KUKA KRL program: nplacestr6RS1.src, nplacestr6RS1.dat

--- nplacestr6RS1.src ---
&ACCESS RVP
&REL 1
&PARAM TEMPLATE = C:\KRC\Roboter\Template\ExpertVorgabe
&PARAM EDITMASK = *
DEF nplacestr6RS1( )
;FOLD INI
  ;FOLD BASISTECH INI
    GLOBAL INTERRUPT DECL 3 WHEN $STOPMESS==TRUE DO IR_STOPM ( )
    INTERRUPT ON 3
    BAS (#INITMOV,0 )
  ;ENDFOLD (BASISTECH INI)
  ;FOLD USER INI
    ;Make your modifications here

  ;ENDFOLD (USER INI)
;ENDFOLD (INI)




SWITCH NumCuring

;*******************************************************
CASE 90613
;*******************************************************
;*** Utilizar para hacer touchup en ptp a continuacion ***;
; 1  Ejecutar Axis_Rob_Move
; 2  Hacer TouchUp en ptp
; 3  Eliminar Axis_Rob_Move y comentarios

Axis_Rob_Move(1.69,-82.8,66.93,14.32,12.14,193,70,50)

;FOLD PTP pWB90613RS1 Vel=100 % PDAT_MESA Tool[10]:AMF1_G1000 Base[14]:BWB2S1;%{PE}%R 5.5.32,%MKUKATPBASIS,%CMOVE,%VPTP,%P 1:PTP, 2:pWB90613RS1, 3:, 5:100, 7:PDAT_MESA
$BWDSTART=FALSE
PDAT_ACT=PPDAT_MESA
FDAT_ACT=FpWB90613RS1
BAS(#PTP_PARAMS,100)
PTP XpWB90613RS1
;ENDFOLD
;*********************************************************;

;***Axis_Rob_Move de ayuda para aproximarse a dejada ***;
; Borrar tras touchup en LIN de dejada
Axis_Rob_Move(-90.22,-57.13,49.23,-5.44,97.37,193.9,20,50)
;*******************************************************;

PTP_OFFS(XP90613RS1, FP90613RS1, 0, -450, 30, 0, 0, 0, #TOOL, 20, 50, 0.0)

Cicle_Grp_M1000 (Inic_Pla_Right)

;***borrar***;
cyltopos(prg_200)
halt
;************;

LIN_OFFS(XP90613RS1, FP90613RS1, 0, 0, 30, 0, 0, 0, #TOOL, 0.1, 50, 0.0)
LIN_OFFS(XP90613RS1, FP90613RS1, 0, 0, 15, 0, 0, 0, #TOOL, 0.1, 50, 0.0)

Cntr_Grp_M1000 (C05C06,RH)

;FOLD LIN P90613RS1 Vel=0.1 m/s LV020Z0 Tool[10]:AMF1_G1000 Base[14]:BWB2S1;%{PE}%R 5.5.32,%MKUKATPBASIS,%CMOVE,%VLIN,%P 1:LIN, 2:P90613RS1, 3:, 5:0.1, 7:V020Z0
$BWDSTART=FALSE
LDAT_ACT=LV020Z0
FDAT_ACT=FP90613RS1
BAS(#CP_PARAMS,0.1)
LIN XP90613RS1
;ENDFOLD

Cntr_Grp_M1000 (AMF09,RLS)
Cyltopos (PRG_51)
Cntr_Grp_M1000 (C07C08,RH)
Cyltopos (PRG_61)
Cntr_Grp_M1000 (AMF10,RLS)
Cntr_Grp_M1000 (C05C06,FREE)
Cntr_Grp_M1000 (C07C08,FREE)
Cyltopos(PRG_88)
LIN_REL{Z -20}#TOOL
Cyltopos (PRG_105)
LIN_REL{Z -30}#TOOL
Cyltopos (PRG_200)

;*** MOVIMIENTOS DE OFFSETS ***;

LIN_OFFS(XP90613RS1, FP90613RS1, 0, 0, -50, 0, 0, 0, #TOOL, 0.3, 50, 0.0)
LIN_OFFS(XP90613RS1, FP90613RS1, 0, -450, -50, 0, 0, 0, #TOOL, 0.3, 50, 0.0)


;******* MEDICION LASER *******;

LIN_OFFS(XPLAS90613RS1_1, FPLAS90613RS1_1, 0, -200, 0, 0, 0, 0, #TOOL, 0.3, 50, 0.0)

cyltopos (prg_61)

;FOLD LIN PLAS90613RS1_1 Vel=0.3 m/s LV020Z0 Tool[10]:AMF1_G1000 Base[14]:BWB2S1;%{PE}%R 5.5.32,%MKUKATPBASIS,%CMOVE,%VLIN,%P 1:LIN, 2:PLAS90613RS1_1, 3:, 5:0.3, 7:V020Z0
$BWDSTART=FALSE
LDAT_ACT=LV020Z0
FDAT_ACT=FPLAS90613RS1_1
BAS(#CP_PARAMS,0.3)
LIN XPLAS90613RS1_1
;ENDFOLD

;Movimimiento de busqueda con laser
;Search( , )

;FOLD LIN PLAS90613RS1_2 Vel=0.3 m/s LV020Z0 Tool[10]:AMF1_G1000 Base[14]:BWB2S1;%{PE}%R 5.5.32,%MKUKATPBASIS,%CMOVE,%VLIN,%P 1:LIN, 2:PLAS90613RS1_2, 3:, 5:0.3, 7:V020Z0
$BWDSTART=FALSE
LDAT_ACT=LV020Z0
FDAT_ACT=FPLAS90613RS1_2
BAS(#CP_PARAMS,0.3)
LIN XPLAS90613RS1_2
;ENDFOLD


;Movimimiento de busqueda con laser
;Search( , )

LIN_OFFS(XPLAS90613RS1_1, FPLAS90613RS1_1, 0, -200, 0, 0, 0, 0, #TOOL, 0.3, 50, 0.0)

;******************************;

;FOLD PTP pWB90613RS1 Vel=100 % PDAT_MESA Tool[10]:AMF1_G1000 Base[14]:BWB2S1;%{PE}%R 5.5.32,%MKUKATPBASIS,%CMOVE,%VPTP,%P 1:PTP, 2:pWB90613RS1, 3:, 5:100, 7:PDAT_MESA
$BWDSTART=FALSE
PDAT_ACT=PPDAT_MESA
FDAT_ACT=FpWB90613RS1
BAS(#PTP_PARAMS,100)
PTP XpWB90613RS1
;ENDFOLD

;*******************************************************
CASE 90615
;*******************************************************
;*** Utilizar para hacer touchup en ptp a continuacion ***;
; 1  Ejecutar Axis_Rob_Move
; 2  Hacer TouchUp en ptp
; 3  Eliminar Axis_Rob_Move y comentarios

Axis_Rob_Move(1.69,-82.8,66.93,14.32,12.14,193,70,50)

;FOLD PTP pWB90615RS1 Vel=100 % PDAT_MESA Tool[10]:AMF1_G1000 Base[14]:BWB2S1;%{PE}%R 5.5.32,%MKUKATPBASIS,%CMOVE,%VPTP,%P 1:PTP, 2:pWB90615RS1, 3:, 5:100, 7:PDAT_MESA
$BWDSTART=FALSE
PDAT_ACT=PPDAT_MESA
FDAT_ACT=FpWB90615RS1
BAS(#PTP_PARAMS,100)
PTP XpWB90615RS1
;ENDFOLD
;*********************************************************;

;***Axis_Rob_Move de ayuda para aproximarse a dejada ***;
; Borrar tras touchup en LIN de dejada
Axis_Rob_Move(-90.22,-57.13,49.23,-5.44,97.37,193.9,20,50)
;*******************************************************;

PTP_OFFS(XP90615RS1, FP90615RS1, 0, -450, 30, 0, 0, 0, #TOOL, 20, 50, 0.0)

Cicle_Grp_M1000 (Inic_Pla_Right)

;***borrar***;
cyltopos(prg_200)
halt
;************;

LIN_OFFS(XP90615RS1, FP90615RS1, 0, 0, 30, 0, 0, 0, #TOOL, 0.1, 50, 0.0)
LIN_OFFS(XP90615RS1, FP90615RS1, 0, 0, 15, 0, 0, 0, #TOOL, 0.1, 50, 0.0)

Cntr_Grp_M1000 (C05C06,RH)

;FOLD LIN P90615RS1 Vel=0.1 m/s LV020Z0 Tool[10]:AMF1_G1000 Base[14]:BWB2S1;%{PE}%R 5.5.32,%MKUKATPBASIS,%CMOVE,%VLIN,%P 1:LIN, 2:P90615RS1, 3:, 5:0.1, 7:V020Z0
$BWDSTART=FALSE
LDAT_ACT=LV020Z0
FDAT_ACT=FP90615RS1
BAS(#CP_PARAMS,0.1)
LIN XP90615RS1
;ENDFOLD

Cntr_Grp_M1000 (AMF09,RLS)
Cyltopos (PRG_51)
Cntr_Grp_M1000 (C07C08,RH)
Cyltopos (PRG_61)
Cntr_Grp_M1000 (AMF10,RLS)
Cntr_Grp_M1000 (C05C06,FREE)
Cntr_Grp_M1000 (C07C08,FREE)
Cyltopos(PRG_88)
LIN_REL{Z -20}#TOOL
Cyltopos (PRG_105)
LIN_REL{Z -30}#TOOL
Cyltopos (PRG_200)

;*** MOVIMIENTOS DE OFFSETS ***;

LIN_OFFS(XP90615RS1, FP90615RS1, 0, 0, -50, 0, 0, 0, #TOOL, 0.3, 50, 0.0)
LIN_OFFS(XP90615RS1, FP90615RS1, 0, -450, -50, 0, 0, 0, #TOOL, 0.3, 50, 0.0)


;******* MEDICION LASER *******;

LIN_OFFS(XPLAS90615RS1_1, FPLAS90615RS1_1, 0, -200, 0, 0, 0, 0, #TOOL, 0.3, 50, 0.0)

cyltopos (prg_61)

;FOLD LIN PLAS90615RS1_1 Vel=0.3 m/s LV020Z0 Tool[10]:AMF1_G1000 Base[14]:BWB2S1;%{PE}%R 5.5.32,%MKUKATPBASIS,%CMOVE,%VLIN,%P 1:LIN, 2:PLAS90615RS1_1, 3:, 5:0.3, 7:V020Z0
$BWDSTART=FALSE
LDAT_ACT=LV020Z0
FDAT_ACT=FPLAS90615RS1_1
BAS(#CP_PARAMS,0.3)
LIN XPLAS90615RS1_1
;ENDFOLD

;Movimimiento de busqueda con laser
;Search( , )

;FOLD LIN PLAS90615RS1_2 Vel=0.3 m/s LV020Z0 Tool[10]:AMF1_G1000 Base[14]:BWB2S1;%{PE}%R 5.5.32,%MKUKATPBASIS,%CMOVE,%VLIN,%P 1:LIN, 2:PLAS90615RS1_2, 3:, 5:0.3, 7:V020Z0
$BWDSTART=FALSE
LDAT_ACT=LV020Z0
FDAT_ACT=FPLAS90615RS1_2
BAS(#CP_PARAMS,0.3)
LIN XPLAS90615RS1_2
;ENDFOLD


;Movimimiento de busqueda con laser
;Search( , )

LIN_OFFS(XPLAS90615RS1_1, FPLAS90615RS1_1, 0, -200, 0, 0, 0, 0, #TOOL, 0.3, 50, 0.0)

;******************************;

;FOLD PTP pWB90615RS1 Vel=100 % PDAT_MESA Tool[10]:AMF1_G1000 Base[14]:BWB2S1;%{PE}%R 5.5.32,%MKUKATPBASIS,%CMOVE,%VPTP,%P 1:PTP, 2:pWB90615RS1, 3:, 5:100, 7:PDAT_MESA
$BWDSTART=FALSE
PDAT_ACT=PPDAT_MESA
FDAT_ACT=FpWB90615RS1
BAS(#PTP_PARAMS,100)
PTP XpWB90615RS1
;ENDFOLD

;*******************************************************
CASE 90617
;*******************************************************
;*** Utilizar para hacer touchup en ptp a continuacion ***;
; 1  Ejecutar Axis_Rob_Move
; 2  Hacer TouchUp en ptp
; 3  Eliminar Axis_Rob_Move y comentarios

Axis_Rob_Move(1.69,-82.8,66.93,14.32,12.14,193,70,50)

;FOLD PTP pWB90617RS1 Vel=100 % PDAT_MESA Tool[10]:AMF1_G1000 Base[14]:BWB2S1;%{PE}%R 5.5.32,%MKUKATPBASIS,%CMOVE,%VPTP,%P 1:PTP, 2:pWB90617RS1, 3:, 5:100, 7:PDAT_MESA
$BWDSTART=FALSE
PDAT_ACT=PPDAT_MESA
FDAT_ACT=FpWB90617RS1
BAS(#PTP_PARAMS,100)
PTP XpWB90617RS1
;ENDFOLD
;*********************************************************;

;***Axis_Rob_Move de ayuda para aproximarse a dejada ***;
; Borrar tras touchup en LIN de dejada
Axis_Rob_Move(-90.22,-57.13,49.23,-5.44,97.37,193.9,20,50)
;*******************************************************;

PTP_OFFS(XP90617RS1, FP90617RS1, 0, -450, 30, 0, 0, 0, #TOOL, 20, 50, 0.0)

Cicle_Grp_M1000 (Inic_Pla_Right)

;***borrar***;
cyltopos(prg_200)
halt
;************;

LIN_OFFS(XP90617RS1, FP90617RS1, 0, 0, 30, 0, 0, 0, #TOOL, 0.1, 50, 0.0)
LIN_OFFS(XP90617RS1, FP90617RS1, 0, 0, 15, 0, 0, 0, #TOOL, 0.1, 50, 0.0)

Cntr_Grp_M1000 (C05C06,RH)

;FOLD LIN P90617RS1 Vel=0.1 m/s LV020Z0 Tool[10]:AMF1_G1000 Base[14]:BWB2S1;%{PE}%R 5.5.32,%MKUKATPBASIS,%CMOVE,%VLIN,%P 1:LIN, 2:P90617RS1, 3:, 5:0.1, 7:V020Z0
$BWDSTART=FALSE
LDAT_ACT=LV020Z0
FDAT_ACT=FP90617RS1
BAS(#CP_PARAMS,0.1)
LIN XP90617RS1
;ENDFOLD

Cntr_Grp_M1000 (AMF09,RLS)
Cyltopos (PRG_51)
Cntr_Grp_M1000 (C07C08,RH)
Cyltopos (PRG_61)
Cntr_Grp_M1000 (AMF10,RLS)
Cntr_Grp_M1000 (C05C06,FREE)
Cntr_Grp_M1000 (C07C08,FREE)
Cyltopos(PRG_88)
LIN_REL{Z -20}#TOOL
Cyltopos (PRG_105)
LIN_REL{Z -30}#TOOL
Cyltopos (PRG_200)

;*** MOVIMIENTOS DE OFFSETS ***;

LIN_OFFS(XP90617RS1, FP90617RS1, 0, 0, -50, 0, 0, 0, #TOOL, 0.3, 50, 0.0)
LIN_OFFS(XP90617RS1, FP90617RS1, 0, -450, -50, 0, 0, 0, #TOOL, 0.3, 50, 0.0)


;******* MEDICION LASER *******;

LIN_OFFS(XPLAS90617RS1_1, FPLAS90617RS1_1, 0, -200, 0, 0, 0, 0, #TOOL, 0.3, 50, 0.0)

cyltopos (prg_61)

;FOLD LIN PLAS90617RS1_1 Vel=0.3 m/s LV020Z0 Tool[10]:AMF1_G1000 Base[14]:BWB2S1;%{PE}%R 5.5.32,%MKUKATPBASIS,%CMOVE,%VLIN,%P 1:LIN, 2:PLAS90617RS1_1, 3:, 5:0.3, 7:V020Z0
$BWDSTART=FALSE
LDAT_ACT=LV020Z0
FDAT_ACT=FPLAS90617RS1_1
BAS(#CP_PARAMS,0.3)
LIN XPLAS90617RS1_1
;ENDFOLD

;Movimimiento de busqueda con laser
;Search( , )

;FOLD LIN PLAS90617RS1_2 Vel=0.3 m/s LV020Z0 Tool[10]:AMF1_G1000 Base[14]:BWB2S1;%{PE}%R 5.5.32,%MKUKATPBASIS,%CMOVE,%VLIN,%P 1:LIN, 2:PLAS90617RS1_2, 3:, 5:0.3, 7:V020Z0
$BWDSTART=FALSE
LDAT_ACT=LV020Z0
FDAT_ACT=FPLAS90617RS1_2
BAS(#CP_PARAMS,0.3)
LIN XPLAS90617RS1_2
;ENDFOLD


;Movimimiento de busqueda con laser
;Search( , )

LIN_OFFS(XPLAS90617RS1_1, FPLAS90617RS1_1, 0, -200, 0, 0, 0, 0, #TOOL, 0.3, 50, 0.0)

;******************************;

;FOLD PTP pWB90617RS1 Vel=100 % PDAT_MESA Tool[10]:AMF1_G1000 Base[14]:BWB2S1;%{PE}%R 5.5.32,%MKUKATPBASIS,%CMOVE,%VPTP,%P 1:PTP, 2:pWB90617RS1, 3:, 5:100, 7:PDAT_MESA
$BWDSTART=FALSE
PDAT_ACT=PPDAT_MESA
FDAT_ACT=FpWB90617RS1
BAS(#PTP_PARAMS,100)
PTP XpWB90617RS1
;ENDFOLD

;*******************************************************
CASE 90619
;*******************************************************
;*** Utilizar para hacer touchup en ptp a continuacion ***;
; 1  Ejecutar Axis_Rob_Move
; 2  Hacer TouchUp en ptp
; 3  Eliminar Axis_Rob_Move y comentarios

Axis_Rob_Move(1.69,-82.8,66.93,14.32,12.14,193,70,50)

;FOLD PTP pWB90619RS1 Vel=100 % PDAT_MESA Tool[10]:AMF1_G1000 Base[14]:BWB2S1;%{PE}%R 5.5.32,%MKUKATPBASIS,%CMOVE,%VPTP,%P 1:PTP, 2:pWB90619RS1, 3:, 5:100, 7:PDAT_MESA
$BWDSTART=FALSE
PDAT_ACT=PPDAT_MESA
FDAT_ACT=FpWB90619RS1
BAS(#PTP_PARAMS,100)
PTP XpWB90619RS1
;ENDFOLD
;*********************************************************;

;***Axis_Rob_Move de ayuda para aproximarse a dejada ***;
; Borrar tras touchup en LIN de dejada
Axis_Rob_Move(-90.22,-57.13,49.23,-5.44,97.37,193.9,20,50)
;*******************************************************;

PTP_OFFS(XP90619RS1, FP90619RS1, 0, -450, 30, 0, 0, 0, #TOOL, 20, 50, 0.0)

Cicle_Grp_M1000 (Inic_Pla_Right)

;***borrar***;
cyltopos(prg_200)
halt
;************;

LIN_OFFS(XP90619RS1, FP90619RS1, 0, 0, 30, 0, 0, 0, #TOOL, 0.1, 50, 0.0)
LIN_OFFS(XP90619RS1, FP90619RS1, 0, 0, 15, 0, 0, 0, #TOOL, 0.1, 50, 0.0)

Cntr_Grp_M1000 (C05C06,RH)

;FOLD LIN P90619RS1 Vel=0.1 m/s LV020Z0 Tool[10]:AMF1_G1000 Base[14]:BWB2S1;%{PE}%R 5.5.32,%MKUKATPBASIS,%CMOVE,%VLIN,%P 1:LIN, 2:P90619RS1, 3:, 5:0.1, 7:V020Z0
$BWDSTART=FALSE
LDAT_ACT=LV020Z0
FDAT_ACT=FP90619RS1
BAS(#CP_PARAMS,0.1)
LIN XP90619RS1
;ENDFOLD

Cntr_Grp_M1000 (AMF09,RLS)
Cyltopos (PRG_51)
Cntr_Grp_M1000 (C07C08,RH)
Cyltopos (PRG_61)
Cntr_Grp_M1000 (AMF10,RLS)
Cntr_Grp_M1000 (C05C06,FREE)
Cntr_Grp_M1000 (C07C08,FREE)
Cyltopos(PRG_88)
LIN_REL{Z -20}#TOOL
Cyltopos (PRG_105)
LIN_REL{Z -30}#TOOL
Cyltopos (PRG_200)

;*** MOVIMIENTOS DE OFFSETS ***;

LIN_OFFS(XP90619RS1, FP90619RS1, 0, 0, -50, 0, 0, 0, #TOOL, 0.3, 50, 0.0)
LIN_OFFS(XP90619RS1, FP90619RS1, 0, -450, -50, 0, 0, 0, #TOOL, 0.3, 50, 0.0)


;******* MEDICION LASER *******;

LIN_OFFS(XPLAS90619RS1_1, FPLAS90619RS1_1, 0, -200, 0, 0, 0, 0, #TOOL, 0.3, 50, 0.0)

cyltopos (prg_61)

;FOLD LIN PLAS90619RS1_1 Vel=0.3 m/s LV020Z0 Tool[10]:AMF1_G1000 Base[14]:BWB2S1;%{PE}%R 5.5.32,%MKUKATPBASIS,%CMOVE,%VLIN,%P 1:LIN, 2:PLAS90619RS1_1, 3:, 5:0.3, 7:V020Z0
$BWDSTART=FALSE
LDAT_ACT=LV020Z0
FDAT_ACT=FPLAS90619RS1_1
BAS(#CP_PARAMS,0.3)
LIN XPLAS90619RS1_1
;ENDFOLD

;Movimimiento de busqueda con laser
;Search( , )

;FOLD LIN PLAS90619RS1_2 Vel=0.3 m/s LV020Z0 Tool[10]:AMF1_G1000 Base[14]:BWB2S1;%{PE}%R 5.5.32,%MKUKATPBASIS,%CMOVE,%VLIN,%P 1:LIN, 2:PLAS90619RS1_2, 3:, 5:0.3, 7:V020Z0
$BWDSTART=FALSE
LDAT_ACT=LV020Z0
FDAT_ACT=FPLAS90619RS1_2
BAS(#CP_PARAMS,0.3)
LIN XPLAS90619RS1_2
;ENDFOLD


;Movimimiento de busqueda con laser
;Search( , )

LIN_OFFS(XPLAS90619RS1_1, FPLAS90619RS1_1, 0, -200, 0, 0, 0, 0, #TOOL, 0.3, 50, 0.0)

;******************************;

;FOLD PTP pWB90619RS1 Vel=100 % PDAT_MESA Tool[10]:AMF1_G1000 Base[14]:BWB2S1;%{PE}%R 5.5.32,%MKUKATPBASIS,%CMOVE,%VPTP,%P 1:PTP, 2:pWB90619RS1, 3:, 5:100, 7:PDAT_MESA
$BWDSTART=FALSE
PDAT_ACT=PPDAT_MESA
FDAT_ACT=FpWB90619RS1
BAS(#PTP_PARAMS,100)
PTP XpWB90619RS1
;ENDFOLD

;*******************************************************
CASE 90621
;*******************************************************
;*** Utilizar para hacer touchup en ptp a continuacion ***;
; 1  Ejecutar Axis_Rob_Move
; 2  Hacer TouchUp en ptp
; 3  Eliminar Axis_Rob_Move y comentarios

Axis_Rob_Move(1.69,-82.8,66.93,14.32,12.14,193,70,50)

;FOLD PTP pWB90621RS1 Vel=100 % PDAT_MESA Tool[10]:AMF1_G1000 Base[14]:BWB2S1;%{PE}%R 5.5.32,%MKUKATPBASIS,%CMOVE,%VPTP,%P 1:PTP, 2:pWB90621RS1, 3:, 5:100, 7:PDAT_MESA
$BWDSTART=FALSE
PDAT_ACT=PPDAT_MESA
FDAT_ACT=FpWB90621RS1
BAS(#PTP_PARAMS,100)
PTP XpWB90621RS1
;ENDFOLD
;*********************************************************;

;***Axis_Rob_Move de ayuda para aproximarse a dejada ***;
; Borrar tras touchup en LIN de dejada
Axis_Rob_Move(-90.22,-57.13,49.23,-5.44,97.37,193.9,20,50)
;*******************************************************;

PTP_OFFS(XP90621RS1, FP90621RS1, 0, -450, 30, 0, 0, 0, #TOOL, 20, 50, 0.0)

Cicle_Grp_M1000 (Inic_Pla_Right)

;***borrar***;
cyltopos(prg_200)
halt
;************;

LIN_OFFS(XP90621RS1, FP90621RS1, 0, 0, 30, 0, 0, 0, #TOOL, 0.1, 50, 0.0)
LIN_OFFS(XP90621RS1, FP90621RS1, 0, 0, 15, 0, 0, 0, #TOOL, 0.1, 50, 0.0)

Cntr_Grp_M1000 (C05C06,RH)

;FOLD LIN P90621RS1 Vel=0.1 m/s LV020Z0 Tool[10]:AMF1_G1000 Base[14]:BWB2S1;%{PE}%R 5.5.32,%MKUKATPBASIS,%CMOVE,%VLIN,%P 1:LIN, 2:P90621RS1, 3:, 5:0.1, 7:V020Z0
$BWDSTART=FALSE
LDAT_ACT=LV020Z0
FDAT_ACT=FP90621RS1
BAS(#CP_PARAMS,0.1)
LIN XP90621RS1
;ENDFOLD

Cntr_Grp_M1000 (AMF09,RLS)
Cyltopos (PRG_51)
Cntr_Grp_M1000 (C07C08,RH)
Cyltopos (PRG_61)
Cntr_Grp_M1000 (AMF10,RLS)
Cntr_Grp_M1000 (C05C06,FREE)
Cntr_Grp_M1000 (C07C08,FREE)
Cyltopos(PRG_88)
LIN_REL{Z -20}#TOOL
Cyltopos (PRG_105)
LIN_REL{Z -30}#TOOL
Cyltopos (PRG_200)

;*** MOVIMIENTOS DE OFFSETS ***;

LIN_OFFS(XP90621RS1, FP90621RS1, 0, 0, -50, 0, 0, 0, #TOOL, 0.3, 50, 0.0)
LIN_OFFS(XP90621RS1, FP90621RS1, 0, -450, -50, 0, 0, 0, #TOOL, 0.3, 50, 0.0)


;******* MEDICION LASER *******;

LIN_OFFS(XPLAS90621RS1_1, FPLAS90621RS1_1, 0, -200, 0, 0, 0, 0, #TOOL, 0.3, 50, 0.0)

cyltopos (prg_61)

;FOLD LIN PLAS90621RS1_1 Vel=0.3 m/s LV020Z0 Tool[10]:AMF1_G1000 Base[14]:BWB2S1;%{PE}%R 5.5.32,%MKUKATPBASIS,%CMOVE,%VLIN,%P 1:LIN, 2:PLAS90621RS1_1, 3:, 5:0.3, 7:V020Z0
$BWDSTART=FALSE
LDAT_ACT=LV020Z0
FDAT_ACT=FPLAS90621RS1_1
BAS(#CP_PARAMS,0.3)
LIN XPLAS90621RS1_1
;ENDFOLD

;Movimimiento de busqueda con laser
;Search( , )

;FOLD LIN PLAS90621RS1_2 Vel=0.3 m/s LV020Z0 Tool[10]:AMF1_G1000 Base[14]:BWB2S1;%{PE}%R 5.5.32,%MKUKATPBASIS,%CMOVE,%VLIN,%P 1:LIN, 2:PLAS90621RS1_2, 3:, 5:0.3, 7:V020Z0
$BWDSTART=FALSE
LDAT_ACT=LV020Z0
FDAT_ACT=FPLAS90621RS1_2
BAS(#CP_PARAMS,0.3)
LIN XPLAS90621RS1_2
;ENDFOLD


;Movimimiento de busqueda con laser
;Search( , )

LIN_OFFS(XPLAS90621RS1_1, FPLAS90621RS1_1, 0, -200, 0, 0, 0, 0, #TOOL, 0.3, 50, 0.0)

;******************************;

;FOLD PTP pWB90621RS1 Vel=100 % PDAT_MESA Tool[10]:AMF1_G1000 Base[14]:BWB2S1;%{PE}%R 5.5.32,%MKUKATPBASIS,%CMOVE,%VPTP,%P 1:PTP, 2:pWB90621RS1, 3:, 5:100, 7:PDAT_MESA
$BWDSTART=FALSE
PDAT_ACT=PPDAT_MESA
FDAT_ACT=FpWB90621RS1
BAS(#PTP_PARAMS,100)
PTP XpWB90621RS1
;ENDFOLD

;*******************************************************
CASE 90623
;*******************************************************
;*** Utilizar para hacer touchup en ptp a continuacion ***;
; 1  Ejecutar Axis_Rob_Move
; 2  Hacer TouchUp en ptp
; 3  Eliminar Axis_Rob_Move y comentarios

Axis_Rob_Move(1.69,-82.8,66.93,14.32,12.14,193,70,50)

;FOLD PTP pWB90623RS1 Vel=100 % PDAT_MESA Tool[10]:AMF1_G1000 Base[14]:BWB2S1;%{PE}%R 5.5.32,%MKUKATPBASIS,%CMOVE,%VPTP,%P 1:PTP, 2:pWB90623RS1, 3:, 5:100, 7:PDAT_MESA
$BWDSTART=FALSE
PDAT_ACT=PPDAT_MESA
FDAT_ACT=FpWB90623RS1
BAS(#PTP_PARAMS,100)
PTP XpWB90623RS1
;ENDFOLD
;*********************************************************;

;***Axis_Rob_Move de ayuda para aproximarse a dejada ***;
; Borrar tras touchup en LIN de dejada
Axis_Rob_Move(-90.22,-57.13,49.23,-5.44,97.37,193.9,20,50)
;*******************************************************;

PTP_OFFS(XP90623RS1, FP90623RS1, 0, -450, 30, 0, 0, 0, #TOOL, 20, 50, 0.0)

Cicle_Grp_M1000 (Inic_Pla_Right)

;***borrar***;
cyltopos(prg_200)
halt
;************;

LIN_OFFS(XP90623RS1, FP90623RS1, 0, 0, 30, 0, 0, 0, #TOOL, 0.1, 50, 0.0)
LIN_OFFS(XP90623RS1, FP90623RS1, 0, 0, 15, 0, 0, 0, #TOOL, 0.1, 50, 0.0)

Cntr_Grp_M1000 (C05C06,RH)

;FOLD LIN P90623RS1 Vel=0.1 m/s LV020Z0 Tool[10]:AMF1_G1000 Base[14]:BWB2S1;%{PE}%R 5.5.32,%MKUKATPBASIS,%CMOVE,%VLIN,%P 1:LIN, 2:P90623RS1, 3:, 5:0.1, 7:V020Z0
$BWDSTART=FALSE
LDAT_ACT=LV020Z0
FDAT_ACT=FP90623RS1
BAS(#CP_PARAMS,0.1)
LIN XP90623RS1
;ENDFOLD

Cntr_Grp_M1000 (AMF09,RLS)
Cyltopos (PRG_51)
Cntr_Grp_M1000 (C07C08,RH)
Cyltopos (PRG_61)
Cntr_Grp_M1000 (AMF10,RLS)
Cntr_Grp_M1000 (C05C06,FREE)
Cntr_Grp_M1000 (C07C08,FREE)
Cyltopos(PRG_88)
LIN_REL{Z -20}#TOOL
Cyltopos (PRG_105)
LIN_REL{Z -30}#TOOL
Cyltopos (PRG_200)

;*** MOVIMIENTOS DE OFFSETS ***;

LIN_OFFS(XP90623RS1, FP90623RS1, 0, 0, -50, 0, 0, 0, #TOOL, 0.3, 50, 0.0)
LIN_OFFS(XP90623RS1, FP90623RS1, 0, -450, -50, 0, 0, 0, #TOOL, 0.3, 50, 0.0)


;******* MEDICION LASER *******;

LIN_OFFS(XPLAS90623RS1_1, FPLAS90623RS1_1, 0, -200, 0, 0, 0, 0, #TOOL, 0.3, 50, 0.0)

cyltopos (prg_61)

;FOLD LIN PLAS90623RS1_1 Vel=0.3 m/s LV020Z0 Tool[10]:AMF1_G1000 Base[14]:BWB2S1;%{PE}%R 5.5.32,%MKUKATPBASIS,%CMOVE,%VLIN,%P 1:LIN, 2:PLAS90623RS1_1, 3:, 5:0.3, 7:V020Z0
$BWDSTART=FALSE
LDAT_ACT=LV020Z0
FDAT_ACT=FPLAS90623RS1_1
BAS(#CP_PARAMS,0.3)
LIN XPLAS90623RS1_1
;ENDFOLD

;Movimimiento de busqueda con laser
;Search( , )

;FOLD LIN PLAS90623RS1_2 Vel=0.3 m/s LV020Z0 Tool[10]:AMF1_G1000 Base[14]:BWB2S1;%{PE}%R 5.5.32,%MKUKATPBASIS,%CMOVE,%VLIN,%P 1:LIN, 2:PLAS90623RS1_2, 3:, 5:0.3, 7:V020Z0
$BWDSTART=FALSE
LDAT_ACT=LV020Z0
FDAT_ACT=FPLAS90623RS1_2
BAS(#CP_PARAMS,0.3)
LIN XPLAS90623RS1_2
;ENDFOLD


;Movimimiento de busqueda con laser
;Search( , )

LIN_OFFS(XPLAS90623RS1_1, FPLAS90623RS1_1, 0, -200, 0, 0, 0, 0, #TOOL, 0.3, 50, 0.0)

;******************************;

;FOLD PTP pWB90623RS1 Vel=100 % PDAT_MESA Tool[10]:AMF1_G1000 Base[14]:BWB2S1;%{PE}%R 5.5.32,%MKUKATPBASIS,%CMOVE,%VPTP,%P 1:PTP, 2:pWB90623RS1, 3:, 5:100, 7:PDAT_MESA
$BWDSTART=FALSE
PDAT_ACT=PPDAT_MESA
FDAT_ACT=FpWB90623RS1
BAS(#PTP_PARAMS,100)
PTP XpWB90623RS1
;ENDFOLD

;*******************************************************
CASE 90625
;*******************************************************
;*** Utilizar para hacer touchup en ptp a continuacion ***;
; 1  Ejecutar Axis_Rob_Move
; 2  Hacer TouchUp en ptp
; 3  Eliminar Axis_Rob_Move y comentarios

Axis_Rob_Move(1.69,-82.8,66.93,14.32,12.14,193,70,50)

;FOLD PTP pWB90625RS1 Vel=100 % PDAT_MESA Tool[10]:AMF1_G1000 Base[14]:BWB2S1;%{PE}%R 5.5.32,%MKUKATPBASIS,%CMOVE,%VPTP,%P 1:PTP, 2:pWB90625RS1, 3:, 5:100, 7:PDAT_MESA
$BWDSTART=FALSE
PDAT_ACT=PPDAT_MESA
FDAT_ACT=FpWB90625RS1
BAS(#PTP_PARAMS,100)
PTP XpWB90625RS1
;ENDFOLD
;*********************************************************;

;***Axis_Rob_Move de ayuda para aproximarse a dejada ***;
; Borrar tras touchup en LIN de dejada
Axis_Rob_Move(-90.22,-57.13,49.23,-5.44,97.37,193.9,20,50)
;*******************************************************;

PTP_OFFS(XP90625RS1, FP90625RS1, 0, -450, 30, 0, 0, 0, #TOOL, 20, 50, 0.0)

Cicle_Grp_M1000 (Inic_Pla_Right)

;***borrar***;
cyltopos(prg_200)
halt
;************;

LIN_OFFS(XP90625RS1, FP90625RS1, 0, 0, 30, 0, 0, 0, #TOOL, 0.1, 50, 0.0)
LIN_OFFS(XP90625RS1, FP90625RS1, 0, 0, 15, 0, 0, 0, #TOOL, 0.1, 50, 0.0)

Cntr_Grp_M1000 (C05C06,RH)

;FOLD LIN P90625RS1 Vel=0.1 m/s LV020Z0 Tool[10]:AMF1_G1000 Base[14]:BWB2S1;%{PE}%R 5.5.32,%MKUKATPBASIS,%CMOVE,%VLIN,%P 1:LIN, 2:P90625RS1, 3:, 5:0.1, 7:V020Z0
$BWDSTART=FALSE
LDAT_ACT=LV020Z0
FDAT_ACT=FP90625RS1
BAS(#CP_PARAMS,0.1)
LIN XP90625RS1
;ENDFOLD

Cntr_Grp_M1000 (AMF09,RLS)
Cyltopos (PRG_51)
Cntr_Grp_M1000 (C07C08,RH)
Cyltopos (PRG_61)
Cntr_Grp_M1000 (AMF10,RLS)
Cntr_Grp_M1000 (C05C06,FREE)
Cntr_Grp_M1000 (C07C08,FREE)
Cyltopos(PRG_88)
LIN_REL{Z -20}#TOOL
Cyltopos (PRG_105)
LIN_REL{Z -30}#TOOL
Cyltopos (PRG_200)

;*** MOVIMIENTOS DE OFFSETS ***;

LIN_OFFS(XP90625RS1, FP90625RS1, 0, 0, -50, 0, 0, 0, #TOOL, 0.3, 50, 0.0)
LIN_OFFS(XP90625RS1, FP90625RS1, 0, -450, -50, 0, 0, 0, #TOOL, 0.3, 50, 0.0)


;******* MEDICION LASER *******;

LIN_OFFS(XPLAS90625RS1_1, FPLAS90625RS1_1, 0, -200, 0, 0, 0, 0, #TOOL, 0.3, 50, 0.0)

cyltopos (prg_61)

;FOLD LIN PLAS90625RS1_1 Vel=0.3 m/s LV020Z0 Tool[10]:AMF1_G1000 Base[14]:BWB2S1;%{PE}%R 5.5.32,%MKUKATPBASIS,%CMOVE,%VLIN,%P 1:LIN, 2:PLAS90625RS1_1, 3:, 5:0.3, 7:V020Z0
$BWDSTART=FALSE
LDAT_ACT=LV020Z0
FDAT_ACT=FPLAS90625RS1_1
BAS(#CP_PARAMS,0.3)
LIN XPLAS90625RS1_1
;ENDFOLD

;Movimimiento de busqueda con laser
;Search( , )

;FOLD LIN PLAS90625RS1_2 Vel=0.3 m/s LV020Z0 Tool[10]:AMF1_G1000 Base[14]:BWB2S1;%{PE}%R 5.5.32,%MKUKATPBASIS,%CMOVE,%VLIN,%P 1:LIN, 2:PLAS90625RS1_2, 3:, 5:0.3, 7:V020Z0
$BWDSTART=FALSE
LDAT_ACT=LV020Z0
FDAT_ACT=FPLAS90625RS1_2
BAS(#CP_PARAMS,0.3)
LIN XPLAS90625RS1_2
;ENDFOLD


;Movimimiento de busqueda con laser
;Search( , )

LIN_OFFS(XPLAS90625RS1_1, FPLAS90625RS1_1, 0, -200, 0, 0, 0, 0, #TOOL, 0.3, 50, 0.0)

;******************************;

;FOLD PTP pWB90625RS1 Vel=100 % PDAT_MESA Tool[10]:AMF1_G1000 Base[14]:BWB2S1;%{PE}%R 5.5.32,%MKUKATPBASIS,%CMOVE,%VPTP,%P 1:PTP, 2:pWB90625RS1, 3:, 5:100, 7:PDAT_MESA
$BWDSTART=FALSE
PDAT_ACT=PPDAT_MESA
FDAT_ACT=FpWB90625RS1
BAS(#PTP_PARAMS,100)
PTP XpWB90625RS1
;ENDFOLD

ENDSWITCH
END

--- nplacestr6RS1.dat ---
DEFDAT nplacestr6RS1
;FOLD EXTERNAL DECLARATIONS;%{PE}%MKUKATPBASIS,%CEXT,%VCOMMON,%P
;FOLD BASISTECH EXT;%{PE}%MKUKATPBASIS,%CEXT,%VEXT,%P
EXT  BAS (BAS_COMMAND  :IN,REAL  :IN )
DECL INT SUCCESS
;ENDFOLD (BASISTECH EXT)
;FOLD USER EXT;%{E}%MKUKATPUSER,%CEXT,%VEXT,%P
;Make here your modifications

;ENDFOLD (USER EXT)
;ENDFOLD (EXTERNAL DECLARATIONS)
DECL E6POS XpWB90613RS1={X 0,Y 0,Z 0,A 0,B 0,C 0,S 2,T 10,E1 0.0,E2 0.0,E3 0.0,E4 0.0,E5 0.0,E6 0.0}
DECL FDAT FpWB90613RS1={TOOL_NO 10,BASE_NO 14,IPO_FRAME #BASE,POINT2[] " ",TQ_STATE FALSE}
;
DECL E6POS XP90613RS1={X 0,Y 0,Z 0,A 0,B 0,C 0,S 2,T 10,E1 0.0,E2 0.0,E3 0.0,E4 0.0,E5 0.0,E6 0.0}
DECL FDAT FP90613RS1={TOOL_NO 10,BASE_NO 14,IPO_FRAME #BASE,POINT2[] " ",TQ_STATE FALSE}
;
DECL E6POS XPLAS90613RS1_1={X 0,Y 0,Z 0,A 0,B 0,C 0,S 2,T 10,E1 0.0,E2 0.0,E3 0.0,E4 0.0,E5 0.0,E6 0.0}
DECL FDAT FPLAS90613RS1_1={TOOL_NO 10,BASE_NO 14,IPO_FRAME #BASE,POINT2[] " ",TQ_STATE FALSE}
DECL E6POS XPLAS90613RS1_2={X 0,Y 0,Z 0,A 0,B 0,C 0,S 2,T 10,E1 0.0,E2 0.0,E3 0.0,E4 0.0,E5 0.0,E6 0.0}
DECL FDAT FPLAS90613RS1_2={TOOL_NO 10,BASE_NO 14,IPO_FRAME #BASE,POINT2[] " ",TQ_STATE FALSE}
;
DECL E6POS XpWB90615RS1={X 0,Y 0,Z 0,A 0,B 0,C 0,S 2,T 10,E1 0.0,E2 0.0,E3 0.0,E4 0.0,E5 0.0,E6 0.0}
DECL FDAT FpWB90615RS1={TOOL_NO 10,BASE_NO 14,IPO_FRAME #BASE,POINT2[] " ",TQ_STATE FALSE}
;
DECL E6POS XP90615RS1={X 0,Y 0,Z 0,A 0,B 0,C 0,S 2,T 10,E1 0.0,E2 0.0,E3 0.0,E4 0.0,E5 0.0,E6 0.0}
DECL FDAT FP90615RS1={TOOL_NO 10,BASE_NO 14,IPO_FRAME #BASE,POINT2[] " ",TQ_STATE FALSE}
;
DECL E6POS XPLAS90615RS1_1={X 0,Y 0,Z 0,A 0,B 0,C 0,S 2,T 10,E1 0.0,E2 0.0,E3 0.0,E4 0.0,E5 0.0,E6 0.0}
DECL FDAT FPLAS90615RS1_1={TOOL_NO 10,BASE_NO 14,IPO_FRAME #BASE,POINT2[] " ",TQ_STATE FALSE}
DECL E6POS XPLAS90615RS1_2={X 0,Y 0,Z 0,A 0,B 0,C 0,S 2,T 10,E1 0.0,E2 0.0,E3 0.0,E4 0.0,E5 0.0,E6 0.0}
DECL FDAT FPLAS90615RS1_2={TOOL_NO 10,BASE_NO 14,IPO_FRAME #BASE,POINT2[] " ",TQ_STATE FALSE}
;
DECL E6POS XpWB90617RS1={X 0,Y 0,Z 0,A 0,B 0,C 0,S 2,T 10,E1 0.0,E2 0.0,E3 0.0,E4 0.0,E5 0.0,E6 0.0}
DECL FDAT FpWB90617RS1={TOOL_NO 10,BASE_NO 14,IPO_FRAME #BASE,POINT2[] " ",TQ_STATE FALSE}
;
DECL E6POS XP90617RS1={X 0,Y 0,Z 0,A 0,B 0,C 0,S 2,T 10,E1 0.0,E2 0.0,E3 0.0,E4 0.0,E5 0.0,E6 0.0}
DECL FDAT FP90617RS1={TOOL_NO 10,BASE_NO 14,IPO_FRAME #BASE,POINT2[] " ",TQ_STATE FALSE}
;
DECL E6POS XPLAS90617RS1_1={X 0,Y 0,Z 0,A 0,B 0,C 0,S 2,T 10,E1 0.0,E2 0.0,E3 0.0,E4 0.0,E5 0.0,E6 0.0}
DECL FDAT FPLAS90617RS1_1={TOOL_NO 10,BASE_NO 14,IPO_FRAME #BASE,POINT2[] " ",TQ_STATE FALSE}
DECL E6POS XPLAS90617RS1_2={X 0,Y 0,Z 0,A 0,B 0,C 0,S 2,T 10,E1 0.0,E2 0.0,E3 0.0,E4 0.0,E5 0.0,E6 0.0}
DECL FDAT FPLAS90617RS1_2={TOOL_NO 10,BASE_NO 14,IPO_FRAME #BASE,POINT2[] " ",TQ_STATE FALSE}
;
DECL E6POS XpWB90619RS1={X 0,Y 0,Z 0,A 0,B 0,C 0,S 2,T 10,E1 0.0,E2 0.0,E3 0.0,E4 0.0,E5 0.0,E6 0.0}
DECL FDAT FpWB90619RS1={TOOL_NO 10,BASE_NO 14,IPO_FRAME #BASE,POINT2[] " ",TQ_STATE FALSE}
;
DECL E6POS XP90619RS1={X 0,Y 0,Z 0,A 0,B 0,C 0,S 2,T 10,E1 0.0,E2 0.0,E3 0.0,E4 0.0,E5 0.0,E6 0.0}
DECL FDAT FP90619RS1={TOOL_NO 10,BASE_NO 14,IPO_FRAME #BASE,POINT2[] " ",TQ_STATE FALSE}
;
DECL E6POS XPLAS90619RS1_1={X 0,Y 0,Z 0,A 0,B 0,C 0,S 2,T 10,E1 0.0,E2 0.0,E3 0.0,E4 0.0,E5 0.0,E6 0.0}
DECL FDAT FPLAS90619RS1_1={TOOL_NO 10,BASE_NO 14,IPO_FRAME #BASE,POINT2[] " ",TQ_STATE FALSE}
DECL E6POS XPLAS90619RS1_2={X 0,Y 0,Z 0,A 0,B 0,C 0,S 2,T 10,E1 0.0,E2 0.0,E3 0.0,E4 0.0,E5 0.0,E6 0.0}
DECL FDAT FPLAS90619RS1_2={TOOL_NO 10,BASE_NO 14,IPO_FRAME #BASE,POINT2[] " ",TQ_STATE FALSE}
;
DECL E6POS XpWB90621RS1={X 0,Y 0,Z 0,A 0,B 0,C 0,S 2,T 10,E1 0.0,E2 0.0,E3 0.0,E4 0.0,E5 0.0,E6 0.0}
DECL FDAT FpWB90621RS1={TOOL_NO 10,BASE_NO 14,IPO_FRAME #BASE,POINT2[] " ",TQ_STATE FALSE}
;
DECL E6POS XP90621RS1={X 0,Y 0,Z 0,A 0,B 0,C 0,S 2,T 10,E1 0.0,E2 0.0,E3 0.0,E4 0.0,E5 0.0,E6 0.0}
DECL FDAT FP90621RS1={TOOL_NO 10,BASE_NO 14,IPO_FRAME #BASE,POINT2[] " ",TQ_STATE FALSE}
;
DECL E6POS XPLAS90621RS1_1={X 0,Y 0,Z 0,A 0,B 0,C 0,S 2,T 10,E1 0.0,E2 0.0,E3 0.0,E4 0.0,E5 0.0,E6 0.0}
DECL FDAT FPLAS90621RS1_1={TOOL_NO 10,BASE_NO 14,IPO_FRAME #BASE,POINT2[] " ",TQ_STATE FALSE}
DECL E6POS XPLAS90621RS1_2={X 0,Y 0,Z 0,A 0,B 0,C 0,S 2,T 10,E1 0.0,E2 0.0,E3 0.0,E4 0.0,E5 0.0,E6 0.0}
DECL FDAT FPLAS90621RS1_2={TOOL_NO 10,BASE_NO 14,IPO_FRAME #BASE,POINT2[] " ",TQ_STATE FALSE}
;
DECL E6POS XpWB90623RS1={X 0,Y 0,Z 0,A 0,B 0,C 0,S 2,T 10,E1 0.0,E2 0.0,E3 0.0,E4 0.0,E5 0.0,E6 0.0}
DECL FDAT FpWB90623RS1={TOOL_NO 10,BASE_NO 14,IPO_FRAME #BASE,POINT2[] " ",TQ_STATE FALSE}
;
DECL E6POS XP90623RS1={X 0,Y 0,Z 0,A 0,B 0,C 0,S 2,T 10,E1 0.0,E2 0.0,E3 0.0,E4 0.0,E5 0.0,E6 0.0}
DECL FDAT FP90623RS1={TOOL_NO 10,BASE_NO 14,IPO_FRAME #BASE,POINT2[] " ",TQ_STATE FALSE}
;
DECL E6POS XPLAS90623RS1_1={X 0,Y 0,Z 0,A 0,B 0,C 0,S 2,T 10,E1 0.0,E2 0.0,E3 0.0,E4 0.0,E5 0.0,E6 0.0}
DECL FDAT FPLAS90623RS1_1={TOOL_NO 10,BASE_NO 14,IPO_FRAME #BASE,POINT2[] " ",TQ_STATE FALSE}
DECL E6POS XPLAS90623RS1_2={X 0,Y 0,Z 0,A 0,B 0,C 0,S 2,T 10,E1 0.0,E2 0.0,E3 0.0,E4 0.0,E5 0.0,E6 0.0}
DECL FDAT FPLAS90623RS1_2={TOOL_NO 10,BASE_NO 14,IPO_FRAME #BASE,POINT2[] " ",TQ_STATE FALSE}
;
DECL E6POS XpWB90625RS1={X 0,Y 0,Z 0,A 0,B 0,C 0,S 2,T 10,E1 0.0,E2 0.0,E3 0.0,E4 0.0,E5 0.0,E6 0.0}
DECL FDAT FpWB90625RS1={TOOL_NO 10,BASE_NO 14,IPO_FRAME #BASE,POINT2[] " ",TQ_STATE FALSE}
;
DECL E6POS XP90625RS1={X 0,Y 0,Z 0,A 0,B 0,C 0,S 2,T 10,E1 0.0,E2 0.0,E3 0.0,E4 0.0,E5 0.0,E6 0.0}
DECL FDAT FP90625RS1={TOOL_NO 10,BASE_NO 14,IPO_FRAME #BASE,POINT2[] " ",TQ_STATE FALSE}
;
DECL E6POS XPLAS90625RS1_1={X 0,Y 0,Z 0,A 0,B 0,C 0,S 2,T 10,E1 0.0,E2 0.0,E3 0.0,E4 0.0,E5 0.0,E6 0.0}
DECL FDAT FPLAS90625RS1_1={TOOL_NO 10,BASE_NO 14,IPO_FRAME #BASE,POINT2[] " ",TQ_STATE FALSE}
DECL E6POS XPLAS90625RS1_2={X 0,Y 0,Z 0,A 0,B 0,C 0,S 2,T 10,E1 0.0,E2 0.0,E3 0.0,E4 0.0,E5 0.0,E6 0.0}
DECL FDAT FPLAS90625RS1_2={TOOL_NO 10,BASE_NO 14,IPO_FRAME #BASE,POINT2[] " ",TQ_STATE FALSE}
;
ENDDAT
